FUNCTION_BLOCK FB_FalliblePublicMock IMPLEMENTS I_FalliblePublic
VAR
    {attribute 'pytmc' := '
        pv: Error
        io: i
        field: DESC TRUE if in error state. FALSE if not.
    '}
    bError : BOOL;
    {attribute 'pytmc' := '
        pv: ErrorMsg
        io: i
        field: DESC Message to aid in debugging if error is true.
    '}
    sErrorMsg : T_MaxString;
END_VAR


METHOD ClearError

bError := FALSE;
sErrorMsg := '';
END_METHOD


METHOD PUBLIC GetError : BOOL

GetError := bError;
END_METHOD


METHOD PUBLIC GetErrorMsg : T_MaxString

GetErrorMsg := sErrorMsg;
END_METHOD


METHOD SetError
VAR_INPUT
    Msg : T_MaxString;
END_VAR

bError := TRUE;
sErrorMsg := Msg;
END_METHOD

END_FUNCTION_BLOCK

(* stored: Version 1.1.0.1
   POU FB_FalliblePublicMock: Id {947f6e32-e79d-44f7-a83f-d8a6d08aee4e}, SpecialFunc None
   Method ClearError: Id {d8486aeb-715f-4b0e-acf6-9d39e9402b09}
   Method GetError: Id {6e6c52b8-fb8e-4710-9fce-38f9b68eb670}
   Method GetErrorMsg: Id {66e09432-f790-40b5-af89-a0d36b1afa52}
   Method SetError: Id {919fbe67-9b4c-417d-af17-87c566e5bae6} *)
